# EPICS substitutions: streamApp/pluginDb/pluginProcess.substitutions
#
# pluginProcess.substitutions
#

file NDProcess.template
{
	{
    PORT            = "Proc\$(N)",
    P               = "$(CAM):",
	R				= "$(PORT):",
    ADDR            = "\$(ADDR=0)",
    TIMEOUT         = "\$(TIMEOUT=1)",
    NDARRAY_PORT    = "\$(PLUGIN_SRC)",
    NDARRAY_ADDR    = "\$(NDARRAY_ADDR=0)",
	}
}
